DATA_BLOCK "Get_Data"
{ S7_Optimized_Access := 'TRUE' }
VERSION : 0.1G
NON_RETAIN
   VAR
      Machine_Speed : Int;
      Pallet_Present : Bool;
      Pallet_Counter : Int;
      Production_Active : Bool;
   END_VAR


BEGIN

END_DATA_BLOCK

